{attribute 'enable_dynamic_creation'}
FUNCTION_BLOCK FB_VialClosed EXTENDS FB_Vial
VAR_INPUT
END_VAR
VAR_OUTPUT
END_VAR
VAR
END_VAR

{attribute 'object_name' := 'FB_init'}
METHOD FB_init : BOOL
VAR_INPUT
	/// if TRUE, the retain variables are initialized (warm start / cold start)
	bInitRetains: BOOL;
	/// if TRUE, the instance afterwards gets moved into the copy code (online change)
	bInCopyCode: BOOL;
END_VAR
eObjectType := E_ObjectType.OBJECTTYPE_VialClosed;
END_METHOD

END_FUNCTION_BLOCK

(* stored: Version 1.1.0.1, ProductVersion 3.1.4022.18
   POU FB_VialClosed: Id {8467fa84-e9b8-4ae2-a3e2-0b46b3f86b50}, SpecialFunc None
   Method FB_init: Id {56f299d8-ac98-4538-9a5a-fb0e8eb758c0} *)
